FUNCTION_BLOCK XtsCollisionAvoidanceControl
VAR_INPUT
END_VAR
VAR_OUTPUT
END_VAR
VAR
	
	AxisGroup			: AXES_GROUP_REF;
	
	LocalState			: BYTE;
	
	GroupEnable			: MC_GroupEnable;
	GroupDisable		: MC_GroupDisable;
	GroupReadStatus		: MC_GroupReadStatus;
	GroupReadError		: MC_GroupReadError;
	GroupReset			: MC_GroupReset;
	GroupAddAxis		: MC_AddAxisToGroup;
	GroupRemoveAxis		: MC_RemoveAxisFromGroup;
	GroupSetOverride	: MC_GroupSetOverride;
	
END_VAR

// NETWORK 1

METHOD AddAxisToGroup : BOOL
VAR_INPUT
	Axis				: AXIS_REF;
	AxisIdInGroup		: UDINT;
END_VAR
GroupAddAxis(AxesGroup := AxisGroup, Axis := Axis, IdentInGroup := UDINT_TO_IDENTINGROUP(AxisIdInGroup));

GroupAddAxis.Execute	:= TRUE;

IF GroupAddAxis.Done THEN
	AddAxisToGroup := TRUE;
END_IF
END_METHOD

METHOD CyclicUpdate : BOOL
VAR_INPUT
END_VAR
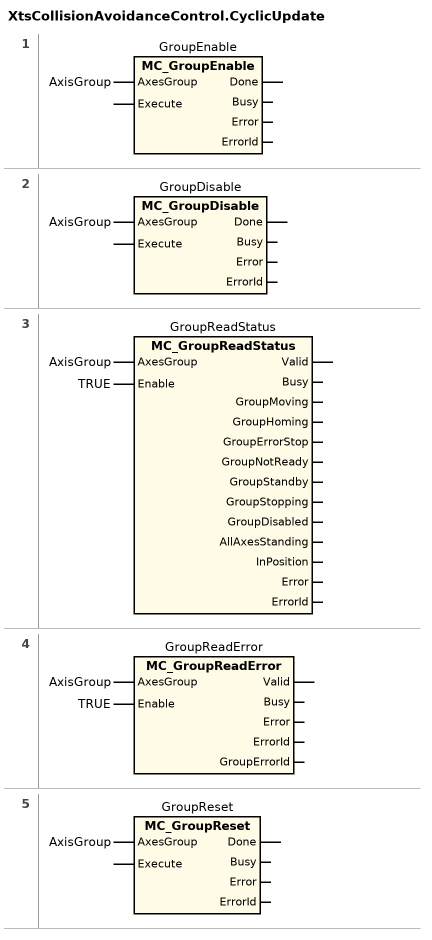
// NETWORK 1
GroupEnable(AxesGroup := AxisGroup); // MC_GroupEnable

// NETWORK 2
GroupDisable(AxesGroup := AxisGroup); // MC_GroupDisable

// NETWORK 3
GroupReadStatus(AxesGroup := AxisGroup, Enable := TRUE); // MC_GroupReadStatus

// NETWORK 4
GroupReadError(AxesGroup := AxisGroup, Enable := TRUE); // MC_GroupReadError

// NETWORK 5
GroupReset(AxesGroup := AxisGroup); // MC_GroupReset
END_METHOD

METHOD DisableGroup : BOOL
VAR_INPUT
END_VAR
END_METHOD

METHOD EnableGroup : BOOL
VAR_INPUT
END_VAR
GroupEnable(AxesGroup := AxisGroup);

GroupEnable.Execute		:= TRUE;

IF GroupEnable.Done THEN
	EnableGroup := TRUE;
END_IF
END_METHOD

METHOD Initialize : BOOL
VAR_INPUT
END_VAR
END_METHOD

METHOD RemoveAxisFromGroup : BOOL
VAR_INPUT
END_VAR
END_METHOD

METHOD ResetGroup : BOOL
VAR_INPUT
END_VAR
GroupReset(AxesGroup := AxisGroup);

GroupReset.Execute := TRUE;

IF GroupReset.Done THEN
	GroupReset.Execute := FALSE;
	ResetGroup := TRUE;
END_IF
END_METHOD

END_FUNCTION_BLOCK

(* stored: Version 1.1.0.1, ProductVersion 3.1.4024.12
   POU XtsCollisionAvoidanceControl: Id {478ffaae-5bbc-4af3-b383-36ee32cae672}, SpecialFunc None
   Folder Power and Utility: Id {57efb649-b87b-4146-95c4-7b48f473b0a4}
   Method AddAxisToGroup: Id {5c73eeda-678c-4cf8-9c55-c194732b85b8}
   Method CyclicUpdate: Id {fe9baa20-02d6-4913-a166-bd502fdcf8b4}
   Method DisableGroup: Id {712bfb01-5961-4f70-aa03-1658a64f03f0}
   Method EnableGroup: Id {d7c4b5bb-e1b2-4fe3-8297-93054f560957}
   Method Initialize: Id {ea229272-ccb3-41f0-95b2-9851cd047b51}
   Method RemoveAxisFromGroup: Id {78d7b7b7-66df-4254-8b3d-9aab699867fb}
   Method ResetGroup: Id {57714453-0127-4882-a694-4a49c1dada25} *)
